(* CODESYS project PLC.project
   Title: PLC
   Version: 0.0.0.0
   Author: Oleksandr

Project tree, tasks and I/O mapping:
  Controller : TM241CEC24T/U, Schneider Electric, order no. TM241CEC24T/U, version 4.0.6.18
    application Application
      task MAST (cyclic, interval 20 ms, priority 15, watchdog 100 ms x 1) calls Main
      global variables GVL
      program Manual [ST]
      program Measure [ST]
      program Main [ST]
      program Auto [ST]
      program Default [ST]
      program Alarms_auto [ST]
      program Alarms_manual [ST]
    DQ : Digital Outputs, Schneider Electric, version 4.0.6.18
        settings: Outputs Usage = 15
        output qwDQ_QW0 : WORD  // QW0
        output qbDQ_QB1 : BYTE  // QB1
    Counters : Counters, Schneider Electric, version 4.0.6.18
    Pulse_Generators : Pulse Generators, Schneider Electric, version 4.0.6.18
        settings: Instance name = 'FreqGen_0'; A output History = 'old=-1 new=0'; Temporary Instance name = 'FreqGen_0'; Instance name = 'FreqGen_1'; A output History = 'old=-1 new=1'; Temporary Instance name = 'FreqGen_1'; Instance name = 'PWM_0'; A output History = 'old=-1 new=2'; Temporary Instance name = 'PWM_0'; Instance name = 'FreqGen_2'; A output History = 'old=-1 new=3'; Temporary Instance name = 'FreqGen_2'
    Cartridge_1 : Cartridge, Schneider Electric, version 4.0.6.18
    IO_Bus : IO bus - TM3, Schneider Electric, version 4.0.6.18
      Module_2 : TM3DQ8R/G, Schneider Electric, order no. TM3DQ8R/G, version 1.0.1.4
          output qbModule_2_QB0 : BYTE  // QB0
      Module_4 : TM3AQ4/G, Schneider Electric, order no. TM3AQ4/G, version 1.0.0.12
          output qiModule_4_QW0 : INT  // QW0
          output qiModule_4_QW1 : INT  // QW1
          output qiModule_4_QW2 : INT  // QW2
          output qiModule_4_QW3 : INT  // QW3
          input  ibModule_4_IBStatusQW0 : BYTE  // IBStatusQW0
          input  ibModule_4_IBStatusQW1 : BYTE  // IBStatusQW1
          input  ibModule_4_IBStatusQW2 : BYTE  // IBStatusQW2
          input  ibModule_4_IBStatusQW3 : BYTE  // IBStatusQW3
      Module_5 : TM3AQ4/G, Schneider Electric, order no. TM3AQ4/G, version 1.0.0.12
          settings: KPI Configuration.KPI Configuration[0] = 16; KPI Configuration.KPI Configuration[1] = 16; KPI Configuration.KPI Configuration[5] = 0; KPI Configuration.KPI Configuration[7] = 0; KPI Configuration.KPI Configuration[12] = 16; KPI Configuration.KPI Configuration[13] = 39; KPI Configuration.KPI Configuration[14] = 16; KPI Configuration.KPI Configuration[15] = 39
          output qiModule_5_QW0 : INT  // QW0
          output qiModule_5_QW1 : INT  // QW1
          output qiModule_5_QW2 : INT  // QW2
          output qiModule_5_QW3 : INT  // QW3
          input  ibModule_5_IBStatusQW0 : BYTE  // IBStatusQW0
          input  ibModule_5_IBStatusQW1 : BYTE  // IBStatusQW1
          input  ibModule_5_IBStatusQW2 : BYTE  // IBStatusQW2
          input  ibModule_5_IBStatusQW3 : BYTE  // IBStatusQW3
      Module_6 : TM3AI8/G, Schneider Electric, order no. TM3AI8/G, version 1.0.0.17
          settings: KPI Configuration.KPI Configuration[0] = 35; KPI Configuration.KPI Configuration[1] = 35; KPI Configuration.KPI Configuration[2] = 35; KPI Configuration.KPI Configuration[3] = 35; KPI Configuration.KPI Configuration[4] = 35; KPI Configuration.KPI Configuration[5] = 35; KPI Configuration.KPI Configuration[6] = 35; KPI Configuration.KPI Configuration[7] = 35; KPI Configuration.KPI Configuration[8] = 160; KPI Configuration.KPI Configuration[9] = 15; KPI Configuration.KPI Configuration[10] = 160; KPI Configuration.KPI Configuration[11] = 15; KPI Configuration.KPI Configuration[12] = 160; KPI Configuration.KPI Configuration[13] = 15; KPI Configuration.KPI Configuration[14] = 160; KPI Configuration.KPI Configuration[15] = 15; KPI Configuration.KPI Configuration[16] = 160; KPI Configuration.KPI Configuration[17] = 15; KPI Configuration.KPI Configuration[18] = 160; KPI Configuration.KPI Configuration[19] = 15; KPI Configuration.KPI Configuration[20] = 160; KPI Configuration.KPI Configuration[21] = 15; KPI Configuration.KPI Configuration[22] = 160; KPI Configuration.KPI Configuration[23] = 15; KPI Configuration.KPI Configuration[24] = 32; KPI Configuration.KPI Configuration[25] = 78; KPI Configuration.KPI Configuration[26] = 32; KPI Configuration.KPI Configuration[27] = 78; KPI Configuration.KPI Configuration[28] = 32; KPI Configuration.KPI Configuration[29] = 78; KPI Configuration.KPI Configuration[30] = 32; KPI Configuration.KPI Configuration[31] = 78; KPI Configuration.KPI Configuration[32] = 32; KPI Configuration.KPI Configuration[33] = 78; KPI Configuration.KPI Configuration[34] = 32; KPI Configuration.KPI Configuration[35] = 78; KPI Configuration.KPI Configuration[36] = 32; KPI Configuration.KPI Configuration[37] = 78; KPI Configuration.KPI Configuration[38] = 32; KPI Configuration.KPI Configuration[39] = 78
          input  iiModule_6_IW0 : INT  // IW0
          input  iiModule_6_IW1 : INT  // IW1
          input  iiModule_6_IW2 : INT  // IW2
          input  iiModule_6_IW3 : INT  // IW3
          input  iiModule_6_IW4 : INT  // IW4
          input  iiModule_6_IW5 : INT  // IW5
          input  iiModule_6_IW6 : INT  // IW6
          input  iiModule_6_IW7 : INT  // IW7
          input  ibModule_6_IBStatusIW0 : BYTE  // IBStatusIW0
          input  ibModule_6_IBStatusIW1 : BYTE  // IBStatusIW1
          input  ibModule_6_IBStatusIW2 : BYTE  // IBStatusIW2
          input  ibModule_6_IBStatusIW3 : BYTE  // IBStatusIW3
          input  ibModule_6_IBStatusIW4 : BYTE  // IBStatusIW4
          input  ibModule_6_IBStatusIW5 : BYTE  // IBStatusIW5
          input  ibModule_6_IBStatusIW6 : BYTE  // IBStatusIW6
          input  ibModule_6_IBStatusIW7 : BYTE  // IBStatusIW7
      Module_1 : TM3DQ8R/G, Schneider Electric, order no. TM3DQ8R/G, version 1.0.1.4
          output qbModule_1_QB0 : BYTE  // QB0
      Module_3 : TM3DQ8T/G, Schneider Electric, order no. TM3DQ8T/G, version 1.0.1.4
          output qbModule_3_QB0 : BYTE  // QB0
    COM_Bus : COM bus, Schneider Electric, version 4.0.6.18
    DI : Digital Inputs, Schneider Electric, version 4.0.6.18
        input  iwDI_IW0 : WORD  // IW0
        input  ibDI_IB1 : BYTE  // IB1
    Ethernet_1 : Ethernet Network, Schneider Electric, version 4.0.6.18
    Serial_Line_1 : Serial line, Schneider Electric, version 4.0.6.18
      SoMachine_Network_Manager : SoMachine-Network Manager, Schneider Electric, version 4.0.0.2
    Serial_Line_2 : Serial line, Schneider Electric, version 4.0.6.18
      Modbus_Manager : Modbus Manager, Schneider Electric, version 4.0.0.2
    CAN_1 : CANopen bus, Schneider Electric, version 4.0.6.18
      CANopen_Optimized : CANopen Performance, Schneider Electric, order no. 1806, version 3.0.1.24
          settings: Enable Sync generation = FALSE; Sync CobID = 126; Heartbeat in Milliseconds = 100; Enable Heartbeat generation = TRUE; Heartbeat Node ID = 101; Can Open Node ID = 101; ConfigVersion = 50659584
        CEBORA_TIG : CEBORA Power Source, CEBORA S.p.A., order no. 0, version Revision=16#00000000, FileVersion=1.2, File=CEBORA_TIG.eds
            settings: General Options.Create all SDOs = TRUE; General Options.Optional Device = TRUE; NODEIDSAVED = 3; SDO Timeout = 1000000; EXPERTSETTINGS = True; Heartbeat-Producer Time = 200; PDO 16#1400.COBID = 16#0203; PDO 16#1401.COBID = 16#0303; PDO 16#1402.COBID = 16#0403; PDO 16#1800.COBID = 16#0183; PDO 16#1800.Inhibit Time = 0; PDO 16#1800.Event Timer = 0; PDO 16#1801.COBID = 16#0283; PDO 16#1801.Inhibit Time = 0; PDO 16#1801.Event Timer = 0; PDO 16#1802.COBID = 16#0383; PDO 16#1802.Inhibit Time = 0; PDO 16#1802.Event Timer = 0; Heartbeat-Consuming1.Heartbeat-Time = 780 ms; DI0_DI7.Subindex = 16#01; DI8_DI15.Subindex = 16#02; DI16_DI23.Subindex = 16#03; DI24_D31.Subindex = 16#04; DI32_DI39.Subindex = 16#05; DI40_DI47.Subindex = 16#06; DI48_DI55.Subindex = 16#07; DI56_DI63.Subindex = 16#08; Analogue Output 1.Subindex = 16#01; Analogue Output 2.Subindex = 16#02; Analogue Output 3.Subindex = 16#03; Analogue Output 4.Subindex = 16#04; Analogue Output 5.Subindex = 16#05; Analogue Output 6.Subindex = 16#06; Analogue Output 7.Subindex = 16#07; Analogue Output 8.Subindex = 16#08; DO0_DO7.Subindex = 16#01; DO8_DO15.Subindex = 16#02; DO16_DO23.Subindex = 16#03; DO24_DO31.Subindex = 16#04; Analogue Input 1.Subindex = 16#01;
              Analogue Input 2.Subindex = 16#02; Analogue Input 3.Subindex = 16#03; Analogue Input 4.Subindex = 16#04; Analogue Input 5.Subindex = 16#05; Analogue Input 6.Subindex = 16#06; Analogue Input 7.Subindex = 16#07; Analogue Input 8.Subindex = 16#08; SDO List.Set Heartbeat Consumer.Index = 16#1016; SDO List.Set Heartbeat Consumer.Subindex = 16#01; SDO List.Set Heartbeat Consumer.Value = 16#007E030C; SDO List.Set Heartbeat Consumer.Size = 32; SDO List.Set Heartbeat Consumer.AbortIfError = FALSE; SDO List.Set Heartbeat Consumer.JumpToLine = FALSE; SDO List.Set Heartbeat Consumer.Line = 0; SDO List.Set Heartbeat Producer.Index = 16#1017; SDO List.Set Heartbeat Producer.Subindex = 16#00; SDO List.Set Heartbeat Producer.Value = 16#000000C8; SDO List.Set Heartbeat Producer.Size = 16; SDO List.Set Heartbeat Producer.AbortIfError = FALSE; SDO List.Set Heartbeat Producer.JumpToLine = FALSE; SDO List.Set Heartbeat Producer.Line = 0; SDO List.DI0_DI7.Index = 16#6200; SDO List.DI0_DI7.Subindex = 16#01; SDO List.DI0_DI7.Value = 0; SDO List.DI0_DI7.Size = 8; SDO List.DI0_DI7.AbortIfError = FALSE; SDO List.DI0_DI7.JumpToLine = FALSE; SDO List.DI0_DI7.Line = 0; SDO List.DI8_DI15.Index = 16#6200; SDO List.DI8_DI15.Subindex = 16#02; SDO List.DI8_DI15.Value = 0; SDO List.DI8_DI15.Size = 8; SDO List.DI8_DI15.AbortIfError = FALSE; SDO List.DI8_DI15.JumpToLine = FALSE; SDO List.DI8_DI15.Line = 0; SDO List.DI16_DI23.Index = 16#6200; SDO List.DI16_DI23.Subindex = 16#03; SDO List.DI16_DI23.Value = 0; SDO List.DI16_DI23.Size = 8; SDO List.DI16_DI23.AbortIfError = FALSE;
              SDO List.DI16_DI23.JumpToLine = FALSE; SDO List.DI16_DI23.Line = 0; SDO List.DI24_D31.Index = 16#6200; SDO List.DI24_D31.Subindex = 16#04; SDO List.DI24_D31.Value = 0; SDO List.DI24_D31.Size = 8; SDO List.DI24_D31.AbortIfError = FALSE; SDO List.DI24_D31.JumpToLine = FALSE; SDO List.DI24_D31.Line = 0; SDO List.DI32_DI39.Index = 16#6200; SDO List.DI32_DI39.Subindex = 16#05; SDO List.DI32_DI39.Value = 16#FF; SDO List.DI32_DI39.Size = 8; SDO List.DI32_DI39.AbortIfError = FALSE; SDO List.DI32_DI39.JumpToLine = FALSE; SDO List.DI32_DI39.Line = 0; SDO List.DI40_DI47.Index = 16#6200; SDO List.DI40_DI47.Subindex = 16#06; SDO List.DI40_DI47.Value = 0; SDO List.DI40_DI47.Size = 8; SDO List.DI40_DI47.AbortIfError = FALSE; SDO List.DI40_DI47.JumpToLine = FALSE; SDO List.DI40_DI47.Line = 0; SDO List.DI48_DI55.Index = 16#6200; SDO List.DI48_DI55.Subindex = 16#07; SDO List.DI48_DI55.Value = 0; SDO List.DI48_DI55.Size = 8; SDO List.DI48_DI55.AbortIfError = FALSE; SDO List.DI48_DI55.JumpToLine = FALSE; SDO List.DI48_DI55.Line = 0; SDO List.DI56_DI63.Index = 16#6200; SDO List.DI56_DI63.Subindex = 16#08; SDO List.DI56_DI63.Value = 0; SDO List.DI56_DI63.Size = 8; SDO List.DI56_DI63.AbortIfError = FALSE; SDO List.DI56_DI63.JumpToLine = FALSE; SDO List.DI56_DI63.Line = 0; SDO List.Analogue Output 1.Index = 16#6411; SDO List.Analogue Output 1.Subindex = 16#01; SDO List.Analogue Output 1.Value = 16#00000000;
              SDO List.Analogue Output 1.Size = 16; SDO List.Analogue Output 1.AbortIfError = FALSE; SDO List.Analogue Output 1.JumpToLine = FALSE; SDO List.Analogue Output 1.Line = 0; SDO List.Analogue Output 2.Index = 16#6411; SDO List.Analogue Output 2.Subindex = 16#02; SDO List.Analogue Output 2.Value = 16#00000000; SDO List.Analogue Output 2.Size = 16; SDO List.Analogue Output 2.AbortIfError = FALSE; SDO List.Analogue Output 2.JumpToLine = FALSE; SDO List.Analogue Output 2.Line = 0; SDO List.Analogue Output 3.Index = 16#6411; SDO List.Analogue Output 3.Subindex = 16#03; SDO List.Analogue Output 3.Value = 16#00000000; SDO List.Analogue Output 3.Size = 16; SDO List.Analogue Output 3.AbortIfError = FALSE; SDO List.Analogue Output 3.JumpToLine = FALSE; SDO List.Analogue Output 3.Line = 0; SDO List.Analogue Output 4.Index = 16#6411; SDO List.Analogue Output 4.Subindex = 16#04; SDO List.Analogue Output 4.Value = 16#00000000; SDO List.Analogue Output 4.Size = 16; SDO List.Analogue Output 4.AbortIfError = FALSE; SDO List.Analogue Output 4.JumpToLine = FALSE; SDO List.Analogue Output 4.Line = 0; SDO List.Analogue Output 5.Index = 16#6411; SDO List.Analogue Output 5.Subindex = 16#05; SDO List.Analogue Output 5.Value = 16#00000000; SDO List.Analogue Output 5.Size = 16; SDO List.Analogue Output 5.AbortIfError = FALSE; SDO List.Analogue Output 5.JumpToLine = FALSE; SDO List.Analogue Output 5.Line = 0; SDO List.Analogue Output 6.Index = 16#6411; SDO List.Analogue Output 6.Subindex = 16#06; SDO List.Analogue Output 6.Value = 16#00000000; SDO List.Analogue Output 6.Size = 16; SDO List.Analogue Output 6.AbortIfError = FALSE; SDO List.Analogue Output 6.JumpToLine = FALSE; SDO List.Analogue Output 6.Line = 0; SDO List.Analogue Output 7.Index = 16#6411;
              SDO List.Analogue Output 7.Subindex = 16#07; SDO List.Analogue Output 7.Value = 16#00000000; SDO List.Analogue Output 7.Size = 16; SDO List.Analogue Output 7.AbortIfError = FALSE; SDO List.Analogue Output 7.JumpToLine = FALSE; SDO List.Analogue Output 7.Line = 0; SDO List.Analogue Output 8.Index = 16#6411; SDO List.Analogue Output 8.Subindex = 16#08; SDO List.Analogue Output 8.Value = 16#00000000; SDO List.Analogue Output 8.Size = 16; SDO List.Analogue Output 8.AbortIfError = FALSE; SDO List.Analogue Output 8.JumpToLine = FALSE; SDO List.Analogue Output 8.Line = 0; ConfigVersion = 50659584
            output Application.CAN_SET_ArcOn : BOOL  // DI0_DI7.Bit0
            output Application.CAN_SET_RobotReady : BOOL  // DI0_DI7.Bit1
            output Application.CAN_SET_OperMode_0 : BOOL  // DI0_DI7.Bit2
            output Application.CAN_SET_OperMode_1 : BOOL  // DI0_DI7.Bit3
            output Application.CAN_SET_OperMode_2 : BOOL  // DI0_DI7.Bit4
            output Application.CAN_SET_AnalogSwap : BOOL  // DI0_DI7.Bit6
            output Application.CAN_SET_ProtocolMode : BOOL  // DI0_DI7.Bit7
            output Application.CAN_SET_GasTest : BOOL  // DI8_DI15.Bit0
            output Application.CAN_SET_WireInching : BOOL  // DI8_DI15.Bit1
            output Application.CAN_SET_WireRetract : BOOL  // DI8_DI15.Bit2
            output Application.CAN_SET_SourceErrReset : BOOL  // DI8_DI15.Bit3
            output Application.CAN_SET_TouchSensing : BOOL  // DI8_DI15.Bit4
            output Application.CAN_SET_BlowTrough : BOOL  // DI8_DI15.Bit5
            output Application.CAN_SET_JOB_0 : BOOL  // DI16_DI23.Bit0
            output Application.CAN_SET_JOB_1 : BOOL  // DI16_DI23.Bit1
            output Application.CAN_SET_JOB_2 : BOOL  // DI16_DI23.Bit2
            output Application.CAN_SET_JOB_3 : BOOL  // DI16_DI23.Bit3
            output Application.CAN_SET_JOB_4 : BOOL  // DI16_DI23.Bit4
            output Application.CAN_SET_JOB_5 : BOOL  // DI16_DI23.Bit5
            output Application.CAN_SET_JOB_6 : BOOL  // DI16_DI23.Bit6
            output Application.CAN_SET_JOB_7 : BOOL  // DI16_DI23.Bit7
            output Application.CAN_SET_WeldSim : BOOL  // DI24_D31.Bit7
            output Application.CAN_SET_AnalogSetDis_0 : BOOL  // DI32_DI39.Bit0
            output Application.CAN_SET_AnalogSetDis_1 : BOOL  // DI32_DI39.Bit1
            output Application.CAN_SET_AnalogSetDis_2 : BOOL  // DI32_DI39.Bit2
            output Application.CAN_SET_AnalogSetDis_3 : BOOL  // DI32_DI39.Bit3
            output Application.CAN_SET_AnalogSetDis_4 : BOOL  // DI32_DI39.Bit4
            output Application.CAN_SET_AnalogSetDis_5 : BOOL  // DI32_DI39.Bit5
            output Application.CAN_SET_DC_AC_Disable : BOOL  // DI40_DI47.Bit0
            output Application.CAN_SET_PLS_Disable : BOOL  // DI40_DI47.Bit3
            output Application.CAN_SET_DC_AC : BOOL  // DI48_DI55.Bit0
            output Application.CAN_SET_PLS : BOOL  // DI48_DI55.Bit3
            output Application.CAN_SET_PilotArc : BOOL  // DI48_DI55.Bit7
            output Application.CAN_SET_WeldCurrent : INT  // Analogue Output 1
            output Application.CAN_SET_WireHighSpd : INT  // Analogue Output 2
            output Application.CAN_SET_PLS_Ratio : INT  // Analogue Output 3
            output Application.CAN_SET_WireLowSpd : INT  // Analogue Output 4
            output Application.CAN_SET_PlasmaGasFlow : INT  // Analogue Output 5
            output Application.CAN_SET_ShieldGasFlow : INT  // Analogue Output 6
            input  Application.CAN_GET_CurrFlow : BOOL  // DO0_DO7.Bit0
            input  Application.CAN_GET_ProcActive : BOOL  // DO0_DO7.Bit2
            input  Application.CAN_GET_MainCurrent : BOOL  // DO0_DO7.Bit3
            input  Application.CAN_GET_CollisProtect : BOOL  // DO0_DO7.Bit4
            input  Application.CAN_GET_PowSourReady : BOOL  // DO0_DO7.Bit5
            input  Application.CAN_GET_Commun_Ready : BOOL  // DO0_DO7.Bit6
            input  Application.CAN_GET_ErrNumber_0 : BOOL  // DO8_DO15.Bit0
            input  Application.CAN_GET_ErrNumber_1 : BOOL  // DO8_DO15.Bit1
            input  Application.CAN_GET_ErrNumber_2 : BOOL  // DO8_DO15.Bit2
            input  Application.CAN_GET_ErrNumber_3 : BOOL  // DO8_DO15.Bit3
            input  Application.CAN_GET_ErrNumber_4 : BOOL  // DO8_DO15.Bit4
            input  Application.CAN_GET_ErrNumber_5 : BOOL  // DO8_DO15.Bit5
            input  Application.CAN_GET_ErrNumber_6 : BOOL  // DO8_DO15.Bit6
            input  Application.CAN_GET_ErrNumber_7 : BOOL  // DO8_DO15.Bit7
            input  Application.CAN_GET_PLS_Sync : BOOL  // DO16_DO23.Bit0
            input  Application.CAN_GET_PilotArc : BOOL  // DO16_DO23.Bit7
            input  Application.CAN_GET_StikingRem : BOOL  // DO24_DO31.Bit0
            input  Application.CAN_GET_WireAvailale : BOOL  // DO24_DO31.Bit3
            input  Application.CAN_GET_WeldVoltage : INT  // Analogue Input 1
            input  Application.CAN_GET_WeldCurrent : INT  // Analogue Input 2
            input  Application.CAN_GET_MotorCurrent : INT  // Analogue Input 3
            input  Application.CAN_GET_WireFeedSPD : INT  // Analogue Input 4
            input  Application.CAN_GET_PlasmaGasFlw : INT  // Analogue Input 5
            input  Application.CAN_GET_ShieldGasFlw : INT  // Analogue Input 6
            unmapped channels: DI0_DI7, DI8_DI15, DI16_DI23, DI24_D31, DI32_DI39, DI40_DI47, DI48_DI55, DI56_DI63, Analogue Output 7, Analogue Output 8, DO0_DO7, DO8_DO15, DO16_DO23, DO24_DO31, Analogue Input 7, Analogue Input 8
*)

// Controller/Application/GVL
VAR_GLOBAL
	IX0_0 AT %IX0.0:BOOL;
	IX0_1 AT %IX0.1:BOOL;
	IX0_2 AT %IX0.2: BOOL;
	IX0_3 AT %IX0.3: BOOL;
	IX0_4 AT %IX0.4: BOOL;
	IX0_5 AT %IX0.5: BOOL;
	IX0_6 AT %IX0.6: BOOL;
	IX0_7 AT %IX0.7: BOOL;
	IX0_8 AT %IX0.8: BOOL;
	
	IW6 AT %IW6:WORD;
	IW7 AT %IW7:WORD;
	IW8 AT %IW8:WORD;
	IW9 AT %IW9:WORD;
	IW10 AT %IW10:WORD;
	IW11 AT %IW11:WORD;
	IW12 AT %IW12:WORD;
	IW13 AT %IW13:WORD;
	
	QX0_4 AT %QX0.4:BOOL;
	QX0_5 AT %QX0.5:BOOL;
	QX0_6 AT %QX0.6:BOOL;
	QX0_7 AT %QX0.7:BOOL;
	QX1_0 AT %QX1.0:BOOL;
	QX1_1 AT %QX1.1:BOOL;
	QX3_0 AT %QX3.0:BOOL;
	QX3_1 AT %QX3.1:BOOL;
	QX3_2 AT %QX3.2:BOOL;
	QX3_3 AT %QX3.3:BOOL;
	QX3_4 AT %QX3.4:BOOL;
	QX3_5 AT %QX3.5:BOOL;
	QX3_6 AT %QX3.6:BOOL;
	QX3_7 AT %QX3.7:BOOL;
	QX4_0 AT %QX4.0:BOOL;
	QX4_1 AT %QX4.1:BOOL;
	QX4_2 AT %QX4.2:BOOL;
	QX4_3 AT %QX4.3:BOOL;
	QX4_4 AT %QX4.4:BOOL;
	QX4_5 AT %QX4.5:BOOL;
	QX4_6 AT %QX4.6:BOOL;
	QX4_7 AT %QX4.7:BOOL;
	QX5_5 AT %QX5.5:BOOL;
	QW7 AT %QW7:WORD;
	QW8 AT %QW8:WORD;
	
	MW4_14:BOOL;
	ExtRestart_State:BOOL;
	
	TON0_M_State:BOOL;
	TON1_M_State:BOOL;
	TON2_M_State:BOOL;
	TON3_M_State:BOOL;
	TON0_A_State:BOOL;
	TON1_A_State:BOOL;
	TON2_A_State:BOOL;
	TON3_A_State:BOOL;
	TON4_A_State:BOOL;
	TON5_A_State:BOOL;
	TON6_A_State:BOOL;
	TON7_A_State:BOOL;
	TON7_1_A_State:BOOL;
	TON7_2_A_State:BOOL;
	TON8_A_State:BOOL;
	TON8_1_A_State:BOOL;
	TON8_2_A_State:BOOL;
	TON9_A_State:BOOL;
	TON10_A_State:BOOL;
	TON11_A_State:BOOL;
	TON11_1_A_State:BOOL;
	TON12_A_State:BOOL;
	TON12_1_A_State:BOOL;
	TON13_State:BOOL;
	TON14_State:BOOL;
	TON15_State:BOOL;
	TON16_Emergency_stop:BOOL;
	TON17_State:BOOL;
	TON17_SW:BOOL;
	TON18_State:BOOL;
	TON18_SW:BOOL;
	TON19_State:BOOL;
	TON20_Emergency_stop:BOOL;
	
	CAN_SET_ArcOn:BOOL;
	CAN_SET_RobotReady:BOOL;
	CAN_SET_OperMode_0:BOOL;
	CAN_SET_OperMode_1:BOOL;
	CAN_SET_OperMode_2:BOOL;
	CAN_SET_AnalogSwap:BOOL;
	CAN_SET_ProtocolMode:BOOL;
	CAN_SET_GasTest:BOOL;
	CAN_SET_WireInching:BOOL;
	CAN_SET_WireRetract:BOOL;
	CAN_SET_SourceErrReset:BOOL;
	CAN_SET_TouchSensing:BOOL;
	CAN_SET_BlowTrough:BOOL;
	CAN_SET_JOB_0:BOOL;
	CAN_SET_JOB_1:BOOL;
	CAN_SET_JOB_2:BOOL;
	CAN_SET_JOB_3:BOOL;
	CAN_SET_JOB_4:BOOL;
	CAN_SET_JOB_5:BOOL;
	CAN_SET_JOB_6:BOOL;
	CAN_SET_JOB_7:BOOL;
	CAN_SET_WeldSim:BOOL;
	CAN_SET_AnalogSetDis_0:BOOL;
	CAN_SET_AnalogSetDis_1:BOOL;
	CAN_SET_AnalogSetDis_2:BOOL;
	CAN_SET_AnalogSetDis_3:BOOL;
	CAN_SET_AnalogSetDis_4:BOOL;
	CAN_SET_AnalogSetDis_5:BOOL;
	CAN_SET_DC_AC_Disable:BOOL;
	CAN_SET_PLS_Disable:BOOL;
	CAN_SET_DC_AC:BOOL;
	CAN_SET_PLS:BOOL;
	CAN_SET_PilotArc:BOOL;
	
	CAN_SET_WeldCurrent:UINT;
	CAN_SET_WireHighSpd:UINT;
	CAN_SET_PLS_Ratio:UINT;
	CAN_SET_WireLowSpd:UINT;
	CAN_SET_PlasmaGasFlow:UINT;
	CAN_SET_ShieldGasFlow:UINT;
	
	CAN_GET_CurrFlow:BOOL;
	CAN_GET_ProcActive:BOOL;
	CAN_GET_MainCurrent:BOOL;
	CAN_GET_CollisProtect:BOOL;
	CAN_GET_PowSourReady:BOOL;
	CAN_GET_Commun_Ready:BOOL;
	CAN_GET_ErrNumber_0:BOOL;
	CAN_GET_ErrNumber_1:BOOL;
	CAN_GET_ErrNumber_2:BOOL;
	CAN_GET_ErrNumber_3:BOOL;
	CAN_GET_ErrNumber_4:BOOL;
	CAN_GET_ErrNumber_5:BOOL;
	CAN_GET_ErrNumber_6:BOOL;
	CAN_GET_ErrNumber_7:BOOL;
	CAN_GET_PLS_Sync:BOOL;
	CAN_GET_PilotArc:BOOL;
	CAN_GET_StikingRem:BOOL;
	CAN_GET_WireAvailale:BOOL;
	
	CAN_GET_WeldVoltage:UINT;
	CAN_GET_WeldCurrent:UINT;
	CAN_GET_MotorCurrent:UINT;
	CAN_GET_WireFeedSPD:UINT;
	CAN_GET_PlasmaGasFlw:UINT;
	CAN_GET_ShieldGasFlw:UINT;
	
	MW110 AT %MW110:WORD;
	MW112 AT %MW112:WORD;
	MW114 AT %MW114:WORD;
	MW116 AT %MW116:WORD;
	MW118 AT %MW118:WORD;
	MW120 AT %MW120:WORD;
	MW122 AT %MW122:WORD;
	MW124 AT %MW124:WORD;
	MW126 AT %MW126:WORD;
	MW128 AT %MW128:WORD;
END_VAR

VAR_GLOBAL RETAIN
	MW0 AT %MW0:WORD;
	MW2 AT %MW2:WORD;
	MW4 AT %MW4:WORD;
	MW6 AT %MW6:WORD;
	MW8 AT %MW8:WORD;
	MW10 AT %MW10:WORD;
	MW12 AT %MW12:WORD;
	MW14 AT %MW14:WORD;
	MW16 AT %MW16:WORD;
	MW18 AT %MW18:WORD;
	MW20 AT %MW20:WORD;
	MW22 AT %MW22:WORD;
	MW24 AT %MW24:WORD;
	MW26 AT %MW26:WORD;
	MW28 AT %MW28:WORD;
	MW30 AT %MW30:WORD;
	MW32 AT %MW32:WORD;
	MW34 AT %MW34:WORD;
	MW36 AT %MW36:WORD;
	MW38 AT %MW38:WORD;
	MW40 AT %MW40:WORD;
	MW44 AT %MW44:WORD;
	MW42 AT %MW42:WORD;
	MW46 AT %MW46:WORD;
	MW48 AT %MW48:WORD;
	MW50 AT %MW50:WORD;
	MW52 AT %MW52:WORD;
	MW54 AT %MW54:WORD;
	MW56 AT %MW56:WORD;
	MW58 AT %MW58:WORD;
	MW60 AT %MW60:WORD;
	MW62 AT %MW62:WORD;
	MW64 AT %MW64:WORD;
	MW66 AT %MW66:WORD;
	MW68 AT %MW68:WORD;
	MW70 AT %MW70:WORD;
	MW72 AT %MW72:WORD;
	MW74 AT %MW74:WORD;
	MW76 AT %MW76:WORD;
	MW78 AT %MW78:WORD;
	MW80 AT %MW80:WORD;
	MW82 AT %MW82:WORD;
	MW84 AT %MW84:WORD;
	MW86 AT %MW86:WORD;
	MW88 AT %MW88:WORD;
	MW90 AT %MW90:WORD;
	MW92 AT %MW92:WORD;
	MW94 AT %MW94:WORD;
	MW96 AT %MW96:WORD;
	MW98 AT %MW98:WORD;
	MW100 AT %MW100:WORD;
	MW102 AT %MW102:WORD;
	
	MD210 AT %MD210:DWORD;
	MD214 AT %MD214:DWORD;
	MD222 AT %MD222:DWORD;
	MD232 AT %MD232:DWORD;
	MD254 AT %MD254:DWORD;
END_VAR

// Controller/Application/Main
PROGRAM Main
VAR
	RTRIG1: R_TRIG;
END_VAR

QX4_7:= TRUE; //Подача сигналу "Керування від ЛПЗР" на Schneider-робота
IF MW0.5 THEN  Alarms_manual(); ELSE Alarms_auto(); END_IF //Аларми
Measure();
RTRIG1(CLK:= NOT(MW0.5));
IF IX0_0 OR RTRIG1.Q THEN Default(); END_IF //Скидання до дефолту
IF MW0.5 THEN  Manual(); ELSE Auto(); END_IF //Ручний/Автоматичний

END_PROGRAM

// Controller/Application/Alarms_manual
PROGRAM Alarms_manual
VAR
	TON13: TON;
	TON14: TON;
	TON15: TON;
	TON16: TON;
	TON19: TON;
	TON20: TON;
END_VAR

//Затримка аналізу аварій
TON19(IN:= MW0.7 OR MW0.9 OR MW0.10 OR MW0.11, PT:= WORD_TO_TIME(MW96), Q=> TON19_State);
//Аларми загальні
IF TON19_State THEN 
	IF IX0_0 THEN MW100:= 1; MW8.1:= TRUE; END_IF //Аларм по грибку
	IF MW18.12 AND MW0.7 AND IX0_8 THEN MW100:= 2; MW8.1:= TRUE; END_IF //Аларм по аварії лазера
	IF MW8.6 AND IW6 < MW80 THEN MW100:= 5; MW8.1:= TRUE; END_IF //Аларм по низькому тиску газу зварювання
	IF MW8.7 AND IW7 < MW82 THEN MW100:= 6; MW8.1:= TRUE; END_IF //Аларм по низькому тиску газу різання
	IF MW8.8 AND IW8 < MW84 THEN MW100:= 7; MW8.1:= TRUE; END_IF //Аларм по низьких витратах газу зварювання
	IF MW8.9 AND IW9 < MW86 THEN MW100:= 8; MW8.1:= TRUE; END_IF //Аларм по низьких витратах газу різання
END_IF
IF MW8.12 AND MW18.8 AND TON19_State AND MW0.9 AND IW12 < MW92 THEN MW100:= 9; MW8.1:= TRUE; END_IF //Аларм по низькому струму різання
IF MW8.13 AND MW18.8 AND TON19_State AND MW0.9 AND IW13 < MW94 THEN MW100:= 10; MW8.1:= TRUE; END_IF //Аларм по низькій напрузі різання
IF MW8.10 AND MW18.8 AND TON19_State AND (MW0.10 OR MW0.11) AND CAN_GET_WeldCurrent < MW88 THEN MW100:= 11; MW8.1:= TRUE; END_IF //Аларм низькому струму звар
IF MW8.11 AND MW18.8 AND TON19_State AND (MW0.10 OR MW0.11) AND CAN_GET_WeldVoltage < MW90 THEN MW100:= 12; MW8.1:= TRUE; END_IF //Аларм по низькій напрузі звар
//Готовність лазера
IF NOT(MW8.1) AND NOT(IX0_0) AND ((MW18.12 AND NOT(IX0_8)) OR NOT(MW18.12)) AND ((MW8.6 AND IW6 >= MW80) OR NOT(MW8.6)) AND ((MW8.7 AND IW7 >= MW82) OR NOT(MW8.7)) THEN 
	MW8.3:= TRUE; ELSE MW8.3:= FALSE; END_IF
//Готовність різання та зварювання
IF NOT(MW8.1) AND NOT(IX0_0) AND ((MW8.6 AND IW6 >= MW80) OR NOT(MW8.6)) AND ((MW8.7 AND IW7 >= MW82) OR NOT(MW8.7)) THEN 
	MW8.4:= TRUE; MW8.5:= TRUE; ELSE MW8.4:= FALSE; MW8.5:= FALSE; END_IF
//Скидання готовностей при виникненні помилки
IF MW8.1 THEN MW8.3:= FALSE; MW8.4:= FALSE; MW8.5:= FALSE; END_IF
//Затримка аварійного вимкнення
TON20(IN:= MW8.1, PT:= WORD_TO_TIME(MW98), Q=> TON20_Emergency_stop);
//Скидання аларму
IF MW8.0 THEN MW100:= 0; MW8.1:= FALSE; END_IF
//Видача готовності шафи керування на робот
IF MW8.3 OR MW8.4 OR MW8.5 THEN QX4_4:= TRUE; ELSE QX4_4:= FALSE; END_IF

END_PROGRAM

// Controller/Application/Alarms_auto
PROGRAM Alarms_auto
VAR
	TON13: TON;
	TON14: TON;
	TON15: TON;
	TON16: TON;
END_VAR

//Затримка аналізу аварій
TON13(IN:= MW34.10, PT:= WORD_TO_TIME(MW96), Q=> TON13_State);
//Затримка аналізу чергової дуги
TON14(IN:= TON1_A_State, PT:= WORD_TO_TIME(MW60), Q=> TON14_State);
//Затримка аналізу основної дуги
TON15(IN:= (MW34.2 AND NOT(MW34.1) AND QX5_5) OR (MW34.1 AND CAN_SET_ArcOn), PT:= WORD_TO_TIME(MW64), Q=> TON15_State);
//Аларми
IF TON13_State THEN
	IF IX0_0 THEN MW100:= 1; MW8.1:= TRUE; END_IF //Аларм по грибку
	IF MW18.12 AND IX0_8 THEN MW100:= 2; MW8.1:= TRUE; END_IF //Аларм по аварії лазера
	IF MW18.13 AND MW34.4 AND NOT(IX0_4) THEN MW100:= 3; MW8.1:= TRUE; END_IF //Аларм по неготовності робота
	IF MW18.14 AND MW34.4 AND IX0_6 THEN MW100:= 4; MW8.1:= TRUE; END_IF //Аларм по аварії робота
	IF MW8.6 AND IW6 < MW80 THEN MW100:= 5; MW8.1:= TRUE; END_IF //Аларм по низькому тиску газу зварювання
	IF MW8.7 AND IW7 < MW82 THEN MW100:= 6; MW8.1:= TRUE; END_IF //Аларм по низькому тиску газу різання
	IF MW8.8 AND IW8 < MW84 THEN MW100:= 7; MW8.1:= TRUE; END_IF //Аларм по низьких витратах газу зварювання
	IF MW8.9 AND IW9 < MW86 THEN MW100:= 8; MW8.1:= TRUE; END_IF //Аларм по низьких витратах газу різання
END_IF
IF MW8.12 AND MW18.8 AND TON13_State AND QX5_5 AND IW12 < MW92 THEN MW100:= 9; MW8.1:= TRUE; END_IF //Аларм по низькому струму різання
IF MW8.13 AND MW18.8 AND TON13_State AND QX5_5 AND IW13 < MW94 THEN MW100:= 10; MW8.1:= TRUE; END_IF //Аларм по низькій напрузі різання
IF MW8.10 AND MW18.8 AND TON13_State AND (CAN_SET_ArcOn OR CAN_SET_PilotArc) AND CAN_GET_WeldCurrent < MW88 THEN MW100:= 11; MW8.1:= TRUE; END_IF //Аларм низькому струму звар
IF MW8.11 AND MW18.8 AND TON13_State AND (CAN_SET_ArcOn OR CAN_SET_PilotArc) AND CAN_GET_WeldVoltage < MW90 THEN MW100:= 12; MW8.1:= TRUE; END_IF //Аларм по низькій напрузі звар
//Контроль на обрив чергової дуги
IF TON14_State AND TON13_State AND MW18.10 AND (CAN_SET_ArcOn OR CAN_SET_PilotArc) AND NOT(MW18.7) THEN MW100:= 13; MW8.1:= TRUE; END_IF
//Контроль на обрив основної дуги
IF TON15_State AND TON13_State AND MW18.11 AND NOT(MW18.8) THEN MW100:= 14; MW8.1:= TRUE; END_IF
//Скидання готовності при виникненні помилки
IF MW8.1 THEN MW8.2:= FALSE; END_IF
//Готовність в автоматі
IF NOT(MW8.1) AND NOT(IX0_0) AND ((MW34.4 AND ((MW18.13 AND IX0_4) OR NOT(MW18.13)) AND ((MW18.14 AND NOT(IX0_6)) OR NOT(MW18.14))) OR NOT(MW34.4)) AND ((MW18.12 AND MW34.00 AND NOT(IX0_8)) OR NOT(MW18.12) OR NOT(MW34.00)) AND ((MW8.6 AND IW6 >= MW80) OR NOT(MW8.6)) AND ((MW8.7 AND IW7 >= MW82) OR NOT(MW8.7)) THEN
	MW8.2:= TRUE; ELSE MW8.2:= FALSE; END_IF
//Затримка аварійного вимкнення
TON16(IN:= MW8.1, PT:= WORD_TO_TIME(MW98), Q=> TON16_Emergency_stop);
//Скидання аларму
IF MW8.0 THEN MW100:= 0; MW8.1:= FALSE; END_IF
QX4_4:= MW8.2; //Видача готовності шафи керування на робот

END_PROGRAM

// Controller/Application/Measure
PROGRAM Measure
VAR
END_VAR

//Дискретні сигнали
MW18.3:= IX0_0;
MW18.4:= IX0_8;
MW18.5:= IX0_4;
MW18.6:= IX0_6;
MW18.9:= IX0_5;
MW18.7:= CAN_GET_PilotArc;
IF QX5_5 AND (CAN_SET_ArcOn OR CAN_SET_PilotArc) THEN MW18.8:= IX0_2 AND CAN_GET_MainCurrent;
ELSIF QX5_5 THEN MW18.8:= IX0_2;
ELSIF CAN_SET_ArcOn OR CAN_SET_PilotArc THEN MW18.8:= CAN_GET_MainCurrent; 
ELSIF NOT(IX0_2) AND NOT(CAN_GET_MainCurrent) THEN MW18.8:= FALSE; END_IF
QX4_5:= MW18.8; //Видача Main current на робот

//Аналогові входи
IF IW12 >= 4800 THEN //Cutting current
	MW114:= IW12;
ELSE
	MW114:= 4000;
END_IF
IF IW13 >= 4500 THEN //Cutting voltage
	MW116:= IW13;
ELSE
	MW116:= 4000;
END_IF
IF IW6 >= 4100 THEN //BP1 pl. wel.
	MW118:= IW6;
ELSE
	MW118:= 4000;
END_IF
IF IW7 >= 4100 THEN //BP2 pl. cut.
	MW120:= IW7;
ELSE
	MW120:= 4000;
END_IF
IF IW8 >= 4100 THEN //FT2 pl. wel.
	MW122:= IW8;
ELSE
	MW122:= 3674;
END_IF
IF IW9 >= 4100 THEN //FT7 pl. cut.
	MW124:= IW9;
ELSE
	MW124:= 3839;
END_IF

//Вимірювання струму зварювання Cebora
IF CAN_GET_WeldCurrent <= 655 THEN
	MW110:= 0;
ELSE
	MW110:= CAN_GET_WeldCurrent;
END_IF

//Вимірювання напруги зварювання Cebora
IF CAN_GET_WeldVoltage <= 5000 THEN
	MW112:= 0;
ELSE
	MW112:= CAN_GET_WeldVoltage;
END_IF

//Вимірювання Cebora plasma gas
IF CAN_GET_PlasmaGasFlw <= 655 THEN
	MW126:= 0;
ELSE
	MW126:= CAN_GET_PlasmaGasFlw;
END_IF

//Вимірювання Cebora shield gas
IF CAN_GET_ShieldGasFlw <= 220 THEN
	MW128:= 0;
ELSE
	MW128:= CAN_GET_ShieldGasFlw;
END_IF

END_PROGRAM

// Controller/Application/Default
PROGRAM Default
VAR
	I: INT;
END_VAR

MW34.10:= FALSE;
MW0.7:= FALSE;
MW0.9:= FALSE;
MW0.10:= FALSE;
MW0.11:= FALSE;
MW4.1:= FALSE;
MW4.2:= FALSE;
MW4.3:= FALSE;
MW4.4:= FALSE;
MW4.5:= FALSE;
MW4.7:= FALSE;
MW4.8:= FALSE;
MW4.9:= FALSE;
MW4.10:= FALSE;
MW4.11:= FALSE;
MW4.12:= FALSE;
MW4.13:= FALSE;
MW4.14:= FALSE;
MW18.1:= FALSE;
MW18.2:= FALSE;
MD210:= 0;
MD214:= 0;
QX0_6:= TRUE;
QX0_7:= TRUE;
QX3_0:= FALSE; 
QX3_1:= FALSE; 
QX3_2:= FALSE; 
QX3_3:= FALSE; 
QX3_4:= FALSE; 
QX3_5:= FALSE; 
QX3_6:= FALSE; 
QX3_7:= FALSE;
QX4_0:= FALSE; 
QX4_1:= FALSE; 
QX4_2:= FALSE; 
QX4_3:= FALSE; 
MD254:= 0;
QX1_0:= FALSE; 
QX1_1:= FALSE; 
MD222:=0; 
MW28:= 0; 
QW8:= 0;
CAN_SET_ArcOn:= FALSE;
CAN_SET_PilotArc:= FALSE;
CAN_SET_WeldCurrent:= 0;
CAN_SET_RobotReady:= FALSE;
QX5_5:= FALSE;
QW7:= 0;
//Конфігурація частотних виходів
FreqGen_0(EN_Enable:= TRUE, F_Enable:= TRUE, EN_Sync:= TRUE, F_Sync:= TRUE, Frequency:= MD210);
FreqGen_1(EN_Enable:= TRUE, F_Enable:= TRUE, EN_Sync:= TRUE, F_Sync:= TRUE, Frequency:= MD214);
FreqGen_2( EN_Enable:= TRUE, F_Enable:= TRUE,  EN_Sync:= TRUE,  F_Sync:= TRUE, Frequency:= MD254);
PWM_0(EN_Enable:= TRUE, F_Enable:= TRUE, EN_Sync:= TRUE, F_Sync:= TRUE,  Frequency:= MD222, Duty:= MW28);

END_PROGRAM

// Controller/Application/Manual
PROGRAM Manual
VAR
	WORD_AS_BIT_1: WORD_AS_BIT;
	TON0: TON;
	TON1: TON;
	TON2: TON;
	TON3: TON;
	TON17: TON;
	TON18: TON;
END_VAR

//Індикація мигання надпису ALARM
TON17(IN:= NOT(TON17_SW), PT:= T#1S, Q=> TON17_State);
TON18(IN:= TON17_SW, PT:= T#1S, Q=> TON18_State);
IF TON17_State THEN TON17_SW:= TRUE; TON18_SW:= FALSE; END_IF
IF TON18_State THEN TON17_SW:= FALSE; TON18_SW:= TRUE; END_IF
IF MW8.1 THEN
	IF TON17_SW THEN TON18_State:= FALSE; MW102:= 1; END_IF	 
	IF TON18_SW THEN TON17_State:= FALSE; MW102:= 0; END_IF
END_IF

//Керування газами
WORD_AS_BIT_1( W:= MW4,B01=> QX3_0, B02=> QX3_1, B03=> QX3_2, B04=> QX3_3, B05=> QX3_4, B07=> QX3_5, B08=> QX3_6, B09=> QX3_7, B10=> QX4_0, B11=> QX4_1, B12=> QX4_2, B13=> QX4_3, B14=>MW4_14);
IF MW4_14 THEN
	MD232:= WORD_TO_DWORD(MW32);
ELSE
	MD232:= 0;
END_IF
FreqGen_2(
	EN_Enable:= TRUE, 
	F_Enable:= TRUE, 
	EN_Sync:= TRUE, 
	F_Sync:= TRUE, 
	Frequency:= MD232);

//Керування двигуном подачі дроту
QX0_4:= MW18.0;
TON0(IN:= MW18.1, PT:= T#1MS, Q=> TON0_M_State);
TON1(IN:= NOT(MW18.1), PT:= T#1MS, Q=> TON1_M_State);
IF MW18.1 THEN
	QX0_6:= FALSE;
END_IF
IF MW18.1 AND TON0_M_State THEN
	MD210:= WORD_TO_DWORD(MW10);
END_IF
IF NOT(MW18.1) THEN
	MD210:= 0;
END_IF
IF NOT(MW18.1) AND TON1_M_State THEN
	QX0_6:= TRUE;
END_IF
FreqGen_0(
	EN_Enable:= TRUE, 
	F_Enable:= TRUE, 
	EN_Sync:= TRUE, 
	F_Sync:= TRUE, 
	Frequency:= MD210);

//Керування двигуном подачі порошку
TON2(IN:= MW18.2, PT:= T#1MS, Q=> TON2_M_State);
TON3(IN:= NOT(MW18.2), PT:= T#1MS, Q=> TON3_M_State);
IF MW18.2 THEN
	QX0_7:= FALSE;
END_IF
IF MW18.2 AND TON2_M_State THEN
	MD214:= WORD_TO_DWORD(MW14);
END_IF
IF NOT(MW18.2) THEN
	MD214:= 0;
END_IF
IF NOT(MW18.2) AND TON3_M_State THEN
	QX0_7:= TRUE;
END_IF
FreqGen_1(
	EN_Enable:= TRUE, 
	F_Enable:= TRUE, 
	EN_Sync:= TRUE, 
	F_Sync:= TRUE, 
	Frequency:= MD214);
	
//Керування лазером
IF MW0.7 OR (MW0.6 AND MW8.3) THEN MW0.8:= FALSE; ELSE MW0.8:= TRUE; END_IF
IF MW0.6 THEN
	QW8:= MW20;
ELSE
	QW8:= 0;
END_IF
IF MW0.7 AND MW8.3 THEN
	QX1_0:= TRUE;
	QX1_1:= TRUE;
	MD222:= WORD_TO_DWORD(MW22);
	MW28:= MW26;
ELSIF NOT(MW0.7) OR TON20_Emergency_stop THEN
	MW0.7:= FALSE;
	QX1_0:= FALSE;
	QX1_1:= FALSE;
	MD222:= 0;
	MW28:= 0;
END_IF
PWM_0(
	EN_Enable:= TRUE, 
	F_Enable:= TRUE, 
	EN_Sync:= TRUE, 
	F_Sync:= TRUE,  
	Frequency:= MD222, 
	Duty:= MW28);
	
//Керування джерелом різання
IF MW0.9 OR (MW0.13 AND MW8.4) THEN MW0.15:= FALSE; ELSE MW0.15:= TRUE; END_IF
IF MW0.13 THEN
	QW7:= MW16;
ELSE 
	QW7:= 0;
END_IF
IF MW0.9 AND MW8.4 THEN
	QX5_5:= TRUE;
ELSIF NOT(MW0.9) OR TON20_Emergency_stop THEN
	MW0.9:= FALSE;
	QX5_5:= FALSE;
END_IF

//Керування джерелом зварювання
IF MW0.10 OR MW0.11 OR (MW0.12 AND MW8.5) THEN MW0.14:= FALSE; ELSE MW0.14:= TRUE; END_IF
CAN_SET_WeldSim:= MW0.0;
CAN_SET_PlasmaGasFlow:= MW24;
CAN_SET_ShieldGasFlow:= MW30;
CAN_SET_OperMode_1:= TRUE;
CAN_SET_OperMode_2:= TRUE;
IF MW0.12 THEN
	CAN_SET_RobotReady:= TRUE;
	CAN_SET_WeldCurrent:= MW12;
ELSE
	CAN_SET_RobotReady:= FALSE;
	CAN_SET_WeldCurrent:= 0;
END_IF
IF MW0.10 AND MW8.5 THEN
	CAN_SET_PilotArc:= TRUE;
	IF MW0.11 AND MW8.5 THEN
		CAN_SET_ArcOn:= TRUE;
	ELSIF NOT(MW0.11) OR TON20_Emergency_stop THEN
		MW0.11:= FALSE;
		CAN_SET_ArcOn:= FALSE;
	END_IF
ELSIF NOT(MW0.10) OR TON20_Emergency_stop THEN
	MW0.10:= FALSE;
	MW0.11:= FALSE;
	CAN_SET_PilotArc:= FALSE;
	CAN_SET_ArcOn:= FALSE;
	MW0.11:= FALSE;
END_IF
//Блок переходу в автомат та видача IN PROGRESS в ручному режимі
IF CAN_SET_ArcOn OR CAN_SET_PilotArc OR QX5_5 OR QX1_0 OR QX1_1 THEN MW8.14:= TRUE; QX4_6:= TRUE; ELSE MW8.14:= FALSE; QX4_6:= FALSE; END_IF

END_PROGRAM

// Controller/Application/Auto
PROGRAM Auto
VAR
	TON1: TON;
	TON4: TON;
	TON2: TON;
	TON0: TON;
	TON7: TON;
	TON8: TON;
	TON7_1: TON;
	TON8_1: TON;
	TON7_2: TON;
	TON8_2: TON;
	TON6: TON;
	TON9: TON;
	TON10: TON;
	TON11: TON;
	TON12: TON;
	TON11_1: TON;
	TON12_1: TON;
	TON17: TON;
	TON18: TON;
END_VAR

//Індикація процесу на кнопці старт/стоп
TON17(IN:= NOT(TON17_SW), PT:= T#1S, Q=> TON17_State);
TON18(IN:= TON17_SW, PT:= T#1S, Q=> TON18_State);
IF TON17_State THEN TON17_SW:= TRUE; TON18_SW:= FALSE; END_IF
IF TON18_State THEN TON17_SW:= FALSE; TON18_SW:= TRUE; END_IF
IF MW34.10 THEN
	MW6:= 1; 
ELSE 
	IF MW34.7 THEN 
		MW6:= 2;
	ELSE
		IF MW8.1 THEN
			IF TON17_SW THEN TON18_State:= FALSE; MW6:= 3; END_IF	 
			IF TON18_SW THEN TON17_State:= FALSE; MW6:= 0; END_IF
		ELSE
			MW6:= 0;
		END_IF
	END_IF
END_IF
//Застереження від повторного зовнішнього старту
IF NOT(IX0_5) THEN ExtRestart_State:= TRUE; END_IF

//Блок Are you sure/Stop
IF MW34.10 THEN MW34.6:= FALSE;
ELSE
	IF NOT(MW34.4) AND MW8.2 THEN MW34.6:= FALSE; 
	ELSIF MW34.4 OR NOT(MW8.2) THEN MW34.6:= TRUE; END_IF
END_IF

//Трігери старт/стоп процесу
IF NOT(MW34.4) THEN
	IF TON16_Emergency_stop THEN MW34.10:= FALSE; END_IF
	IF MW34.8 THEN 
		IF MW34.10 THEN MW34.10:= FALSE;
		ELSIF MW8.2 THEN MW34.5:= TRUE; END_IF
		MW34.8:= FALSE;
	END_IF
ELSE
	IF (MW34.10 AND MW34.8) OR NOT(IX0_5) OR TON16_Emergency_stop THEN MW34.10:= FALSE; MW34.8:= FALSE; END_IF
	IF IX0_5 AND ExtRestart_State AND MW8.2 THEN MW34.10:= TRUE; ExtRestart_State:=FALSE; END_IF
END_IF

//Цикл автоматичного режиму
QX0_4:= FALSE; //Напрямок двигуна дроту
QX0_5:= FALSE; //Напрямок двигуна порошку
TON1(IN:= MW34.10, PT:= WORD_TO_TIME(MW56), Q=> TON1_A_State);
//Конфігурація частотних виходів
FreqGen_0(EN_Enable:= TRUE, F_Enable:= TRUE, EN_Sync:= TRUE, F_Sync:= TRUE, Frequency:= MD210);
FreqGen_1(EN_Enable:= TRUE, F_Enable:= TRUE, EN_Sync:= TRUE, F_Sync:= TRUE, Frequency:= MD214);
FreqGen_2( EN_Enable:= TRUE, F_Enable:= TRUE,  EN_Sync:= TRUE,  F_Sync:= TRUE, Frequency:= MD254);
PWM_0(EN_Enable:= TRUE, F_Enable:= TRUE, EN_Sync:= TRUE, F_Sync:= TRUE,  Frequency:= MD222, Duty:= MW28);
//Задання попередніх параметрів зварювання до старту
CAN_SET_OperMode_1:= TRUE;
CAN_SET_OperMode_2:= TRUE;
CAN_SET_WeldSim:= MW34.3;
CAN_SET_PlasmaGasFlow:= MW44;
CAN_SET_ShieldGasFlow:= MW46;
//START
IF MW34.10 THEN 
	MW34.7:= TRUE; //In Process start
	//Керування подачею дроту та порошку
	TON7(IN:= MW2.13 AND (((MW34.1 OR MW34.2) AND MW18.8) OR (MW34.0 AND NOT(MW34.1) AND NOT(MW34.2))), PT:= WORD_TO_TIME(MW68), Q=> TON7_A_State);
	TON8(IN:= MW2.14 AND (((MW34.1 OR MW34.2) AND MW18.8) OR (MW34.0 AND NOT(MW34.1) AND NOT(MW34.2))), PT:= WORD_TO_TIME(MW70), Q=> TON8_A_State);
	TON7_1 (IN:= TON7_A_State, PT:= T#1MS, Q=> TON7_1_A_State);
	TON8_1 (IN:= TON8_A_State, PT:= T#1MS, Q=> TON8_1_A_State);
	TON7_2 (IN:= NOT(MW2.13), PT:= T#1MS, Q=> TON7_2_A_State);
	TON8_2 (IN:= NOT(MW2.14), PT:= T#1MS, Q=> TON8_2_A_State);
	IF TON7_A_State THEN QX0_6:= FALSE; END_IF
	IF TON7_A_State AND TON7_1_A_State THEN MD210:= WORD_TO_DWORD(MW50); END_IF
	IF TON8_A_State THEN QX0_7:= FALSE; END_IF
	IF TON8_A_State AND TON8_1_A_State THEN MD214:= WORD_TO_DWORD(MW52); END_IF
	IF NOT(MW2.13) THEN MD210:= 0; END_IF
	IF NOT(MW2.14) THEN MD214:= 0; END_IF
	IF TON7_2_A_State THEN QX0_6:= TRUE; END_IF
	IF TON8_2_A_State THEN QX0_7:= TRUE; END_IF
	//Керування газами
	IF MW2.1 THEN 
		IF NOT(MW18.8) THEN QX3_1:= TRUE; END_IF
	ELSE QX3_1:= FALSE; END_IF
	IF MW2.6 THEN
		IF NOT(MW18.8) THEN QX3_6:= TRUE; END_IF
	ELSE QX3_6:= FALSE; END_IF
	QX3_0:= MW2.0; QX3_3:= MW2.3; QX3_4:= MW2.4; QX3_5:= MW2.5; QX4_1:= MW2.9; QX4_2:= MW2.10; QX4_3:= MW2.11;
	IF MW2.12 THEN MD254:= WORD_TO_DWORD(MW54); ELSE MD254:= 0; END_IF
	IF MW2.2 THEN
		IF MW18.8 THEN QX3_2:= TRUE; END_IF
	ELSE QX3_2:= FALSE; END_IF
	IF MW2.7 THEN
		IF MW18.8 THEN QX3_7:= TRUE; END_IF
	ELSE QX3_7:= FALSE; END_IF
	IF MW2.8 THEN
		IF MW18.8 THEN QX4_0:= TRUE; END_IF
	ELSE QX4_0:= FALSE; END_IF
	TON6(IN:= MW18.8, PT:= WORD_TO_TIME(MW66), Q=> TON6_A_State);
	IF TON6_A_State THEN QX3_1:= FALSE; QX3_6:= FALSE; END_IF
	//Керування лазером
	TON2(IN:= TON1_A_State AND MW34.0 AND ((NOT(MW34.1) AND NOT(MW34.2)) OR ((MW34.1 OR MW34.2) AND MW18.8)), PT:= WORD_TO_TIME(MW58), Q=> TON2_A_State);
	IF MW34.0 AND TON2_A_State THEN QW8:= MW36; END_IF
	TON0(IN:= MW34.0 AND TON2_A_State, PT:= T#20MS, Q=> TON0_A_State);
	IF TON0_A_State THEN QX1_0:= TRUE; QX1_1:= TRUE; MD222:= WORD_TO_DWORD(MW38); MW28:= MW40;
	ELSE QX1_0:= FALSE; QX1_1:= FALSE; MD222:=0; MW28:= 0; QW8:= 0; END_IF
	//Керування джерелом зварювання
	TON4(IN:= CAN_GET_PilotArc, PT:= WORD_TO_TIME(MW62), Q=> TON4_A_State);
	CAN_SET_RobotReady:= TRUE;
	IF MW34.1 THEN 
		CAN_SET_WeldCurrent:= MW42;
		IF TON1_A_State THEN CAN_SET_PilotArc:= TRUE; END_IF
		IF TON4_A_State THEN CAN_SET_ArcOn:= TRUE; END_IF
	ELSE
		CAN_SET_ArcOn:= FALSE;
		CAN_SET_PilotArc:= FALSE;
		CAN_SET_WeldCurrent:= 0;	
	END_IF
	//Керування джерелом різання
	IF MW34.2 THEN
		QW7:= MW48;
		IF TON1_A_State = TRUE THEN QX5_5:= TRUE; END_IF
	ELSE
		QX5_5:= FALSE;
		QW7:= 0;
	END_IF
ELSE
//STOP
	//Керування джерелом зварювання
	CAN_SET_ArcOn:= FALSE;
	CAN_SET_PilotArc:= FALSE;
	CAN_SET_WeldCurrent:= 0;
	CAN_SET_RobotReady:= FALSE;
	//Керування джерелом різання
	QX5_5:= FALSE;
	QW7:= 0;
END_IF
//Керування подачею дроту та порошку
TON11(IN:= NOT(MW34.10), PT:= WORD_TO_TIME(MW76), Q=> TON11_A_State);
TON11_1(IN:= TON11_A_State, PT:= T#1MS, Q=> TON11_1_A_State);
TON12(IN:= NOT(MW34.10), PT:= WORD_TO_TIME(MW78), Q=> TON12_A_State);
TON12_1(IN:= TON12_A_State, PT:= T#1MS, Q=> TON12_1_A_State);
IF TON11_A_State THEN MD210:= 0; END_IF
IF TON11_1_A_State THEN QX0_6:= TRUE; END_IF
IF TON12_A_State THEN MD214:= 0; END_IF
IF TON12_1_A_State THEN QX0_7:= TRUE; END_IF
//Керування газами
TON10(IN:= NOT(MW34.10), PT:= WORD_TO_TIME(MW74), Q=> TON10_A_State);
IF TON10_A_State THEN 
	QX3_0:= FALSE; QX3_1:= FALSE; QX3_2:= FALSE; QX3_3:= FALSE; QX3_4:= FALSE; QX3_5:= FALSE; QX3_6:= FALSE; QX3_7:= FALSE;
	QX4_0:= FALSE; QX4_1:= FALSE; QX4_2:= FALSE; QX4_3:= FALSE; MD254:= 0;
END_IF
//Керування лазером
TON9(IN:= NOT(MW34.10), PT:= WORD_TO_TIME(MW72), Q=> TON9_A_State);
IF TON9_A_State THEN QX1_0:= FALSE; QX1_1:= FALSE; MD222:=0; MW28:= 0; QW8:= 0; END_IF
//In Process stop
IF TON9_A_State AND TON10_A_State AND TON11_A_State AND TON12_A_State THEN MW34.7:= FALSE; END_IF
QX4_6:= MW34.7; //Видача In progress на робот

END_PROGRAM
